DATA_BLOCK "Axis_FB_DB"
{ S7_Optimized_Access := 'FALSE' }
VERSION : 0.1
// ATTRIBUTES
// AUTO_NUMBER = False
// BLOCK_NUMBER = 2200
// END_ATTRIBUTES
"Axis_FB"

BEGIN

END_DATA_BLOCK

